PROGRAM MAIN
VAR
END_VAR

P_Tc3DALI_EL6821();

END_PROGRAM

(* stored: Version 1.1.0.1, ProductVersion 3.1.4024.16
   POU MAIN: Id {aa7f191c-d870-4535-afb2-19166f3694bc}, SpecialFunc None *)
